FUNCTION_BLOCK State1 EXTENDS AbstractState

METHOD Handle : BOOL
fbTON(IN := TRUE, PT := T#7s);
IF fbTON.Q THEN
	LogString(sString := 'Timer in State 1 fired. Changing State to State 2.');
	ipStatehandler.SetState(eNewState := E_STATES.eState2);
	fbTON(IN := FALSE);
END_IF
END_METHOD

END_FUNCTION_BLOCK

(* stored: Version 1.1.0.1, ProductVersion 3.1.4024.3
   POU State1: Id {a962195b-254c-4618-bc5a-9f5f69aff458}, SpecialFunc None
   Method Handle: Id {c219679e-7cd0-4c1d-90b7-e3a9d29faa22} *)
